COMM SMOVL C00533 BC00533 V=100.0 PL=0  +MOVJ EC00533
COMM SREFP 1 C00534 BC00534  +REFP EC00534
COMM SREFP 2 C00535 BC00535  +REFP EC00535
COMM MACRO1 MJ#(0) ARGF0
COMM ARCON
COMM SMOVL C00536 BC00536 V=10.0  +MOVJ EC00536
COMM SMOVL C00537 BC00537 V=10.0  +MOVJ EC00537
COMM SMOVL C00538 BC00538 V=10.0  +MOVJ EC00538
COMM ARCOF
COMM SMOVL C00539 BC00539 V=400.0  +MOVJ EC00539
COMM SMOVL C00540 BC00540 V=1000.0  +MOVJ EC00540
COMM SFTOF3D
'Path W1887
SFTOF3D
SFTON3D P023
MOVJ C00541 BC00541 VJ=100.00  +MOVJ EC00541 VJ=100.00
SMOVL C00542 BC00542 V=400.0  +MOVJ EC00542
SMOVL C00543 BC00543 V=100.0 PL=0  +MOVJ EC00543
SREFP 1 C00544 BC00544  +REFP EC00544
SREFP 2 C00545 BC00545  +REFP EC00545
MACRO1 MJ#(0) ARGF9
ARCON
SMOVL C00546 BC00546 V=10.0  +MOVJ EC00546
ARCOF
SMOVL C00547 BC00547 V=400.0  +MOVJ EC00547
SMOVL C00548 BC00548 V=1000.0  +MOVJ EC00548
SFTOF3D
MOVJ C00549 BC00549 VJ=100.00  +MOVJ EC00549 VJ=100.00
MOVJ C00550 BC00550 VJ=100.00  +MOVJ EC00550 VJ=100.00
MOVJ C00551 BC00551 VJ=100.00  +MOVJ EC00551 VJ=100.00
'2
MOVJ C00552 BC00552 VJ=100.00  +MOVJ EC00552 VJ=100.00
MOVJ C00553 BC00553 VJ=100.00  +MOVJ EC00553 VJ=20.00
MOVJ C00554 BC00554 VJ=100.00  +MOVJ EC00554 VJ=100.00
'Path W1888
SFTOF3D
SFTON3D P021
MOVJ C00555 BC00555 VJ=15.00  +MOVJ EC00555 VJ=100.00
SMOVL C00556 BC00556 V=400.0  +MOVJ EC00556
SMOVL C00557 BC00557 V=133.3 PL=0  +MOVJ EC00557
SREFP 1 C00558 BC00558  +REFP EC00558
SREFP 2 C00559 BC00559  +REFP EC00559
MACRO1 MJ#(0) ARGF14
ARCON
SMOVL C00560 BC00560 V=10.0  +MOVJ EC00560
ARCOF
SMOVL C00561 BC00561 V=166.7  +MOVJ EC00561
SMOVL C00562 BC00562 V=166.7  +MOVJ EC00562
MACRO1 MJ#(0) ARGF14
SMOVL C00563 BC00563 V=133.3 PL=0  +MOVJ EC00563
ARCON
SMOVL C00564 BC00564 V=10.0  +MOVJ EC00564
ARCOF
SMOVL C00565 BC00565 V=400.0  +MOVJ EC00565
SMOVL C00566 BC00566 V=1000.0  +MOVJ EC00566
SMOVL C00567 BC00567 V=1000.0  +MOVJ EC00567
SFTOF3D
MOVJ C00568 BC00568 VJ=50.00  +MOVJ EC00568 VJ=20.00
MOVJ C00569 BC00569 VJ=100.00  +MOVJ EC00569 VJ=100.00
'Path W1889
SFTOF3D
SFTON3D P021
MOVJ C00570 BC00570 VJ=100.00  +MOVJ EC00570 VJ=100.00
MOVJ C00571 BC00571 VJ=100.00  +MOVJ EC00571 VJ=100.00
SMOVL C00572 BC00572 V=400.0  +MOVJ EC00572
SMOVL C00573 BC00573 V=133.3 PL=0  +MOVJ EC00573
SREFP 1 C00574 BC00574  +REFP EC00574
SREFP 2 C00575 BC00575  +REFP EC00575
MACRO1 MJ#(0) ARGF14
ARCON
SMOVL C00576 BC00576 V=10.0  +MOVJ EC00576
ARCOF
SMOVL C00577 BC00577 V=166.7  +MOVJ EC00577
SMOVL C00578 BC00578 V=166.7  +MOVJ EC00578
SMOVL C00579 BC00579 V=166.7 PL=0  +MOVJ EC00579
ARCON
SMOVL C00580 BC00580 V=10.0  +MOVJ EC00580
ARCOF
SMOVL C00581 BC00581 V=400.0  +MOVJ EC00581
SMOVL C00582 BC00582 V=1000.0  +MOVJ EC00582
SMOVL C00583 BC00583 V=1000.0  +MOVJ EC00583
SFTOF3D
MOVJ C00584 BC00584 VJ=100.00  +MOVJ EC00584 VJ=20.00
MOVJ C00585 BC00585 VJ=100.00  +MOVJ EC00585 VJ=100.00
MOVJ C00586 BC00586 VJ=100.00  +MOVJ EC00586 VJ=100.00
MOVJ C00587 BC00587 VJ=100.00  +MOVJ EC00587 VJ=100.00
MOVJ C00588 BC00588 VJ=100.00  +MOVJ EC00588 VJ=100.00
'3
'Path W1890
SFTOF3D
SFTON3D P023
MOVJ C00589 BC00589 VJ=100.00  +MOVJ EC00589 VJ=100.00
'BRAKUJACY ELEMENT
COMM SMOVL C00590 BC00590 V=400.0  +MOVJ EC00590
COMM SMOVL C00591 BC00591 V=100.0 PL=0  +MOVJ EC00591
COMM SREFP 1 C00592 BC00592  +REFP EC00592
COMM SREFP 2 C00593 BC00593  +REFP EC00593
COMM MACRO1 MJ#(0) ARGF0
COMM ARCON
COMM SMOVL C00594 BC00594 V=10.0  +MOVJ EC00594
COMM SMOVL C00595 BC00595 V=10.0  +MOVJ EC00595
COMM SMOVL C00596 BC00596 V=10.0  +MOVJ EC00596
COMM ARCOF
COMM SMOVL C00597 BC00597 V=400.0  +MOVJ EC00597
COMM SMOVL C00598 BC00598 V=1000.0  +MOVJ EC00598
SFTOF3D
'Path W1891
SFTOF3D
SFTON3D P023
MOVJ C00599 BC00599 VJ=100.00  +MOVJ EC00599 VJ=100.00
SMOVL C00600 BC00600 V=400.0  +MOVJ EC00600
SMOVL C00601 BC00601 V=133.3 PL=0  +MOVJ EC00601
SREFP 1 C00602 BC00602  +REFP EC00602
SREFP 2 C00603 BC00603  +REFP EC00603
MACRO1 MJ#(0) ARGF14
ARCON
SMOVL C00604 BC00604 V=11.7  +MOVJ EC00604
ARCOF
SMOVL C00605 BC00605 V=400.0  +MOVJ EC00605
SMOVL C00606 BC00606 V=1000.0  +MOVJ EC00606
SFTOF3D
MOVJ C00607 BC00607 VJ=100.00  +MOVJ EC00607 VJ=100.00
MOVJ C00608 BC00608 VJ=100.00  +MOVJ EC00608 VJ=20.00
MOVJ C00609 BC00609 VJ=100.00  +MOVJ EC00609 VJ=100.00
MOVJ C00610 BC00610 VJ=100.00  +MOVJ EC00610 VJ=20.00
MOVJ C00611 BC00611 VJ=100.00  +MOVJ EC00611 VJ=100.00
MOVJ C00612 BC00612 VJ=100.00  +MOVJ EC00612 VJ=100.00
'4
'Path W1892
SFTOF3D
SFTON3D P022
MOVJ C00613 BC00613 VJ=100.00  +MOVJ EC00613 VJ=20.00
SMOVL C00614 BC00614 V=400.0  +MOVJ EC00614
SMOVL C00615 BC00615 V=133.3 PL=0  +MOVJ EC00615
SREFP 1 C00616 BC00616  +REFP EC00616
SREFP 2 C00617 BC00617  +REFP EC00617
MACRO1 MJ#(0) ARGF14
ARCON
SMOVL C00618 BC00618 V=10.0  +MOVJ EC00618
ARCOF
SMOVL C00619 BC00619 V=400.0  +MOVJ EC00619
SMOVL C00620 BC00620 V=1000.0  +MOVJ EC00620
SFTOF3D
'Path W1893
SFTOF3D
SFTON3D P022
MOVJ C00621 BC00621 VJ=20.00  +MOVJ EC00621 VJ=100.00
SMOVL C00622 BC00622 V=400.0  +MOVJ EC00622
SMOVL C00623 BC00623 V=133.3 PL=0  +MOVJ EC00623
SREFP 1 C00624 BC00624  +REFP EC00624
SREFP 2 C00625 BC00625  +REFP EC00625
MACRO1 MJ#(0) ARGF14
ARCON
SMOVL C00626 BC00626 V=10.0  +MOVJ EC00626
ARCOF
SMOVL C00627 BC00627 V=400.0  +MOVJ EC00627
SMOVL C00628 BC00628 V=1000.0  +MOVJ EC00628
SFTOF3D
MOVJ C00629 BC00629 VJ=100.00  +MOVJ EC00629 VJ=100.00
MOVJ C00630 BC00630 VJ=100.00  +MOVJ EC00630 VJ=100.00
'6
'Path W1895
SFTOF3D
SFTON3D P022
MOVJ C00631 BC00631 VJ=40.00  +MOVJ EC00631 VJ=100.00
SMOVL C00632 BC00632 V=400.0  +MOVJ EC00632
SMOVL C00633 BC00633 V=133.3 PL=0  +MOVJ EC00633
SREFP 1 C00634 BC00634  +REFP EC00634
SREFP 2 C00635 BC00635  +REFP EC00635
MACRO1 MJ#(0) ARGF14
ARCON
SMOVL C00636 BC00636 V=11.7  +MOVJ EC00636
ARCOF
SMOVL C00637 BC00637 V=166.7  +MOVJ EC00637
SMOVL C00638 BC00638 V=166.7  +MOVJ EC00638
SMOVL C00639 BC00639 V=166.7 PL=0  +MOVJ EC00639
ARCON
SMOVL C00640 BC00640 V=11.7  +MOVJ EC00640
ARCOF
SMOVL C00641 BC00641 V=400.0  +MOVJ EC00641
SMOVL C00642 BC00642 V=1000.0  +MOVJ EC00642
SFTOF3D
MOVJ C00643 BC00643 VJ=100.00  +MOVJ EC00643 VJ=100.00
'Path W1896
SFTOF3D
SFTON3D P022
MOVJ C00644 BC00644 VJ=50.00  +MOVJ EC00644 VJ=100.00
SMOVL C00645 BC00645 V=400.0  +MOVJ EC00645
SMOVL C00646 BC00646 V=133.3 PL=0  +MOVJ EC00646
SREFP 1 C00647 BC00647  +REFP EC00647
SREFP 2 C00648 BC00648  +REFP EC00648
MACRO1 MJ#(0) ARGF14
ARCON
SMOVL C00649 BC00649 V=12.5  +MOVJ EC00649
ARCOF
SMOVL C00650 BC00650 V=400.0  +MOVJ EC00650
SMOVL C00651 BC00651 V=1000.0  +MOVJ EC00651
SFTOF3D
'7
'Path W1897
SFTOF3D
SFTON3D P022
MOVJ C00652 BC00652 VJ=100.00  +MOVJ EC00652 VJ=100.00
SMOVL C00653 BC00653 V=400.0  +MOVJ EC00653
SMOVL C00654 BC00654 V=133.3 PL=0  +MOVJ EC00654
SREFP 1 C00655 BC00655  +REFP EC00655
SREFP 2 C00656 BC00656  +REFP EC00656
MACRO1 MJ#(0) ARGF14
ARCON
SMOVL C00657 BC00657 V=12.5  +MOVJ EC00657
ARCOF
SMOVL C00658 BC00658 V=400.0  +MOVJ EC00658
SMOVL C00659 BC00659 V=1000.0  +MOVJ EC00659
SMOVL C00660 BC00660 V=1000.0  +MOVJ EC00660
SFTOF3D
MOVJ C00661 BC00661 VJ=100.00  +MOVJ EC00661 VJ=100.00
'Path W1898
SFTOF3D
SFTON3D P022
MOVJ C00662 BC00662 VJ=100.00  +MOVJ EC00662 VJ=100.00
SMOVL C00663 BC00663 V=400.0  +MOVJ EC00663
SMOVL C00664 BC00664 V=133.3 PL=0  +MOVJ EC00664
SREFP 1 C00665 BC00665  +REFP EC00665
SREFP 2 C00666 BC00666  +REFP EC00666
MACRO1 MJ#(0) ARGF14
ARCON
SMOVL C00667 BC00667 V=12.5  +MOVJ EC00667
ARCOF
SMOVL C00668 BC00668 V=400.0  +MOVJ EC00668
SMOVL C00669 BC00669 V=1000.0  +MOVJ EC00669
MOVJ C00670 BC00670 VJ=100.00  +MOVJ EC00670 VJ=20.00
MOVJ C00671 BC00671 VJ=100.00  +MOVJ EC00671 VJ=20.00
MOVJ C00672 BC00672 VJ=100.00  +MOVJ EC00672 VJ=20.00
MOVJ C00673 BC00673 VJ=100.00  +MOVJ EC00673 VJ=20.00
MOVJ C00674 BC00674 VJ=100.00  +MOVJ EC00674 VJ=100.00
SFTOF3D
END
